(*

.. <legal notes>

legal notes
=================
| SPDX-FileCopyrightText: © 2026 Oleksandr Tiutyk <trofimich@gmail.com>
| SPDX-License-Identifier: LGPL-3.0-only
| For details check: LGPL-3.0-only_

.. _LGPL-3.0-only: https://www.gnu.org/licenses/lgpl-3.0.en.html

.. </legal notes>

*)

INTERFACE IStaticCollection EXTENDS ICollection

{attribute 'monitoring' := 'call'}
PROPERTY FINAL Full : BOOL
GET
END_GET
END_PROPERTY

END_INTERFACE

(* stored: Version 1.1.0.1
   Itf IStaticCollection: Id {b02c8d8f-c22c-45ac-a0ed-0bf87e149440}
   Property Full: Id {952bd918-a9f4-44e8-8700-3a7257de7e67}
   Get Get: Id {2f32c8d9-bf5b-4e61-a47d-d06aeea8028a} *)
